// TIA Portal V20 export
FUNCTION_BLOCK "CalledInPreInterpolator"   // FB223, LAD
// stored: Access Published, MemoryReserve 100, Namespace Unit1.Em1, SetENOAutomatically false
BEGIN

REGION Network 2
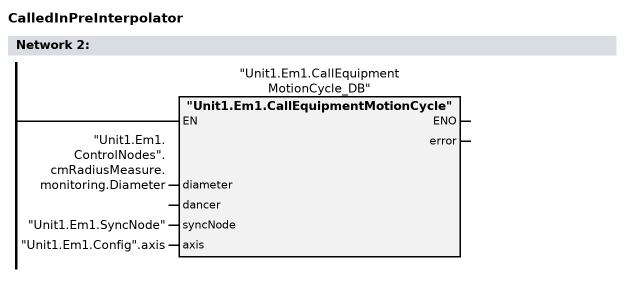
   RUNG wire#powerrail
      "Unit1.Em1.CallEquipmentMotionCycle_DB"(diameter := "Unit1.Em1.ControlNodes".cmRadiusMeasure.monitoring.Diameter, dancer :=, syncNode := "Unit1.Em1.SyncNode", axis := "Unit1.Em1.Config".axis, error =>)
   END_RUNG
   // the same network as SCL:
   "Unit1.Em1.CallEquipmentMotionCycle_DB"(diameter := "Unit1.Em1.ControlNodes".cmRadiusMeasure.monitoring.Diameter,   // "Unit1.Em1.CallEquipmentMotionCycle"
                           syncNode := "Unit1.Em1.SyncNode",
                           axis := "Unit1.Em1.Config".axis);
END_REGION
END_FUNCTION_BLOCK
